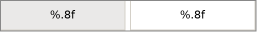
VISUALIZATION VISU_ConfigLREAL8Entry  // 257x32
VAR_IN_OUT
    active : LREAL;
    editable : LREAL;
END_VAR
    Textfield (0,0 125x30), "%.8f", text variable: active, input disabled if: TRUE
    Textfield (130,0 125x30), "%.8f", text variable: editable, colour toggle: editable <> active
        OnMouseClick: write the text variable via Default
END_VISUALIZATION

(* stored: Version 1.1.0.1, ProductVersion 3.1.0.36
   Visu VISU_ConfigLREAL8Entry: Id {340b4516-6a66-4770-8ecb-84d57b98eab3} *)
